PROGRAM Visu
VAR
	Visu_Baum_0: Visu_Baum;
	INT_TRIG_0: INT_TRIG;
	Visu_DayNight_0: Visu_DayNight;
END_VAR

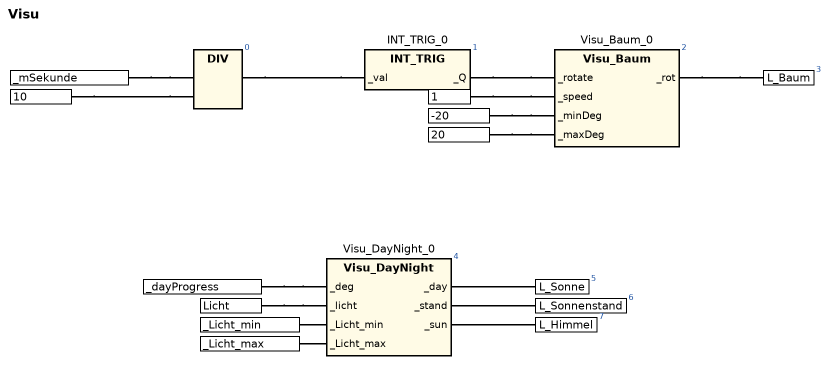
INT_TRIG_0(_val := _mSekunde / 10); // INT_TRIG
Visu_Baum_0(_rotate := INT_TRIG_0._Q, _speed := 1, _minDeg := -20, _maxDeg := 20); // Visu_Baum
L_Baum := Visu_Baum_0._rot;
Visu_DayNight_0(_deg := _dayProgress, _licht := Licht, _Licht_min := _Licht_min, _Licht_max := _Licht_max); // Visu_DayNight
L_Sonne := Visu_DayNight_0._day;
L_Sonnenstand := Visu_DayNight_0._stand;
L_Himmel := Visu_DayNight_0._sun;

END_PROGRAM

(* stored: Version 1.1.0.1, ProductVersion 3.1.4018.5
   POU Visu: Id {641df978-9063-436b-b681-a2092d379665}, SpecialFunc None *)
